INTERFACE I_NumericDatatype EXTENDS I_Datatype

PROPERTY PUBLIC ABSTRACT IsFloat : BOOL
GET
END_GET
END_PROPERTY

PROPERTY PUBLIC IsSigned : BOOL
GET
END_GET
END_PROPERTY

END_INTERFACE

(* stored: Version 1.1.0.1, ProductVersion 3.1.4024.12
   Itf I_NumericDatatype: Id {c5136485-18cb-0c27-1610-72d0069748a7}
   Property IsFloat: Id {9bede2f9-2ecb-08b8-0e06-7ab6bbed3a31}
   Get Get: Id {146766da-1f5a-0441-23e8-b20a0c39604d}
   Property IsSigned: Id {02e02b37-ecdb-04bb-2d74-84539d10b5de}
   Get Get: Id {3712da92-a2e3-07b1-3bec-97a3c6968dd8} *)
